// TIA Portal V20 export
FUNCTION "CallManualOperationLines_Unit1" : Void   // FC69, LAD
// stored: SetENOAutomatically false
   VAR_TEMP
      StatusEm : Array[0..7] of Struct
         Status : Array[0..45] of Word;
      END_STRUCT;
      errorIDEm : Array[0..7] of Struct
         errorID : Array[0..45] of Word;
      END_STRUCT;
      disableUnit1 : Bool;
      TempAxisCommands : "LBC_typeAxis64PosManualCommands";
      TempAxisMonitoring : "LBC_typeAxis64PosProcessValues";
      TempSoftCam : Array[0..8] of "LER_typeSoftCamParameter";
   END_VAR
   VAR CONSTANT
      MECHANIC_NAME_ENABLE : Bool;
   END_VAR
BEGIN

REGION Network 1: Unit 1 Enable Manual Operation
   // Condition to disable manual operation lines in Unit 1
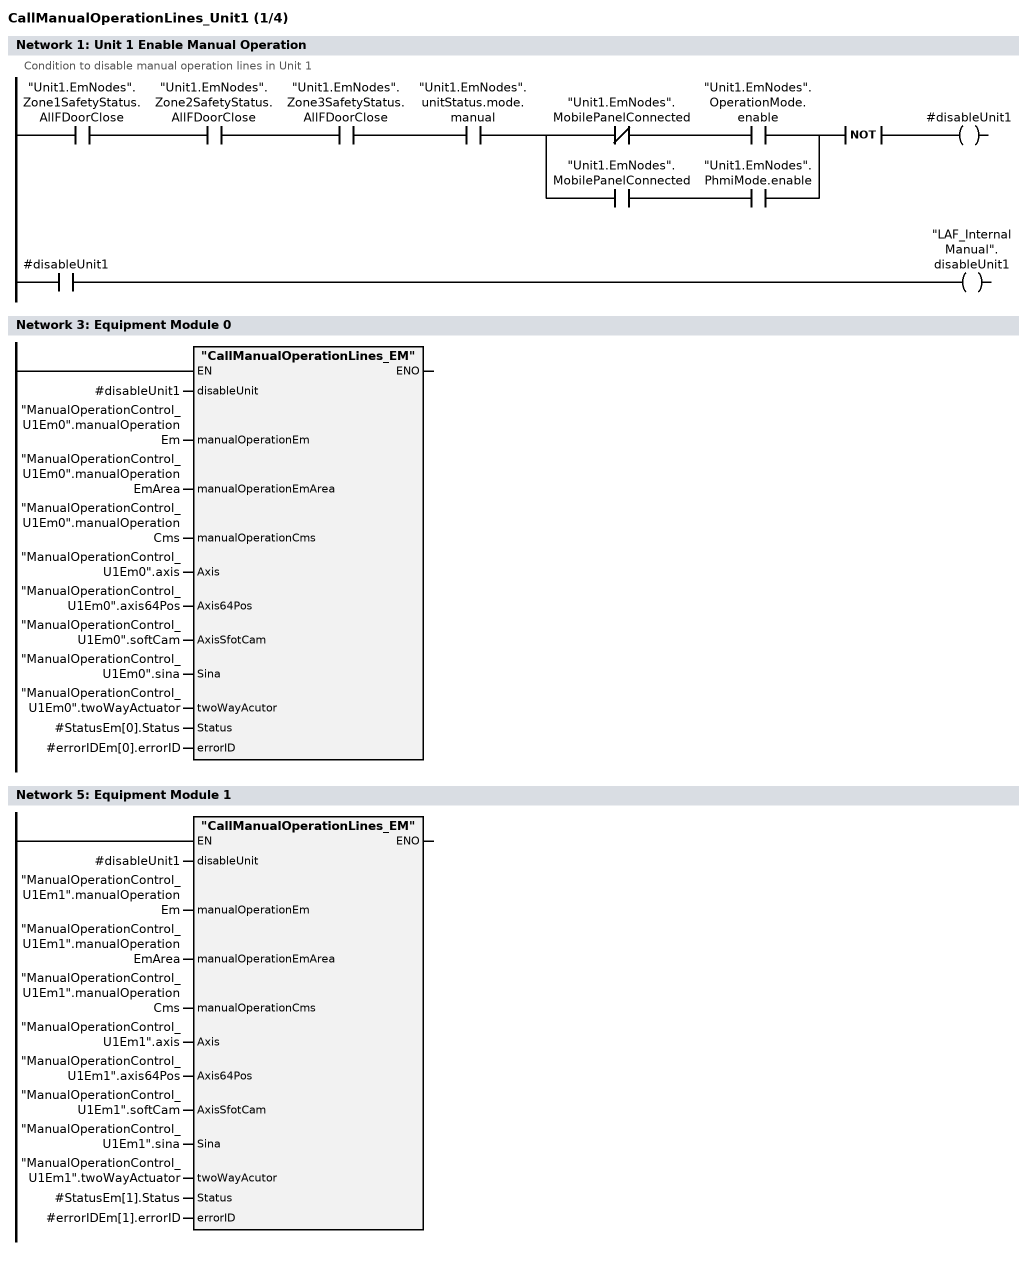
   RUNG wire#powerrail
      Contact( "Unit1.EmNodes".Zone1SafetyStatus.AllFDoorClose )
      Contact( "Unit1.EmNodes".Zone2SafetyStatus.AllFDoorClose )
      Contact( "Unit1.EmNodes".Zone3SafetyStatus.AllFDoorClose )
      Contact( "Unit1.EmNodes".unitStatus.mode.manual )
      wire#w1
      I_Contact( "Unit1.EmNodes".MobilePanelConnected )
      Contact( "Unit1.EmNodes".OperationMode.enable )
      wire#w2
      Not()
      Coil( #disableUnit1 )
   END_RUNG
   RUNG wire#w1
      Contact( "Unit1.EmNodes".MobilePanelConnected )
      Contact( "Unit1.EmNodes".PhmiMode.enable )
   END_RUNG wire#w2
   RUNG wire#powerrail
      Contact( #disableUnit1 )
      Coil( "LAF_InternalManual".disableUnit1 )
   END_RUNG
   // the same network as SCL:
   #disableUnit1 := NOT ("Unit1.EmNodes".Zone1SafetyStatus.AllFDoorClose AND "Unit1.EmNodes".Zone2SafetyStatus.AllFDoorClose AND "Unit1.EmNodes".Zone3SafetyStatus.AllFDoorClose AND "Unit1.EmNodes".unitStatus.mode.manual AND ((NOT "Unit1.EmNodes".MobilePanelConnected AND "Unit1.EmNodes".OperationMode.enable) OR ("Unit1.EmNodes".MobilePanelConnected AND "Unit1.EmNodes".PhmiMode.enable)));
   "LAF_InternalManual".disableUnit1 := #disableUnit1;
END_REGION

REGION Network 2 (SCL): Equipment Module 0 Cms Mapping
   REGION Input Mapping
       // Axis
       "ManualOperationControl_U1Em0".axis[1].monitoring := "Unit1.Em0.HmiInterface".cmUnWinderAxisB.monitoring;

       // TwoWayActuator
       "ManualOperationControl_U1Em0".twoWayActuator[1].monitoring := "Unit1.Em0.HmiInterface".cmAirShaftOnOff.monitoring;
       "ManualOperationControl_U1Em0".twoWayActuator[2].monitoring := "Unit1.Em0.HmiInterface".cmExpelFwdBwd.monitoring;
   END_REGION


   REGION Output Mapping
       // Axis
       "CallManualOperationLines_ServoCommands"(ManualOperationControl := "ManualOperationControl_U1Em0".axis[1].commands,
                                                HmiInterface => "Unit1.Em0.HmiInterface".cmUnWinderAxisB.commands);

       // TwoWayActuator
       "Unit1.Em0.HmiInterface".cmAirShaftOnOff.commands := "ManualOperationControl_U1Em0".twoWayActuator[1].commands;
       "Unit1.Em0.HmiInterface".cmExpelFwdBwd.commands := "ManualOperationControl_U1Em0".twoWayActuator[2].commands;
   END_REGION
END_REGION

REGION Network 3: Equipment Module 0
   RUNG wire#powerrail
      "CallManualOperationLines_EM"(disableUnit := #disableUnit1, manualOperationEm := "ManualOperationControl_U1Em0".manualOperationEm, manualOperationEmArea := "ManualOperationControl_U1Em0".manualOperationEmArea, manualOperationCms := "ManualOperationControl_U1Em0".manualOperationCms, Axis := "ManualOperationControl_U1Em0".axis, Axis64Pos := "ManualOperationControl_U1Em0".axis64Pos, AxisSfotCam := "ManualOperationControl_U1Em0".softCam, Sina := "ManualOperationControl_U1Em0".sina, twoWayAcutor := "ManualOperationControl_U1Em0".twoWayActuator, Status := #StatusEm[0].Status, errorID := #errorIDEm[0].errorID)
   END_RUNG
   // the same network as SCL:
   "CallManualOperationLines_EM"(disableUnit := #disableUnit1,
                           manualOperationEm := "ManualOperationControl_U1Em0".manualOperationEm,
                           manualOperationEmArea := "ManualOperationControl_U1Em0".manualOperationEmArea,
                           manualOperationCms := "ManualOperationControl_U1Em0".manualOperationCms,
                           Axis := "ManualOperationControl_U1Em0".axis,
                           Axis64Pos := "ManualOperationControl_U1Em0".axis64Pos,
                           AxisSfotCam := "ManualOperationControl_U1Em0".softCam,
                           Sina := "ManualOperationControl_U1Em0".sina,
                           twoWayAcutor := "ManualOperationControl_U1Em0".twoWayActuator,
                           Status := #StatusEm[0].Status,
                           errorID := #errorIDEm[0].errorID);
END_REGION

REGION Network 4 (SCL): Equipment Module 1 Cms Mapping
   REGION Input Mapping
       // Axis
       "ManualOperationControl_U1Em1".axis[1].monitoring := "Unit1.Em1.HmiInterface".cmUnWinderAxisB.monitoring;

       // TwoWayActuator
       "ManualOperationControl_U1Em1".twoWayActuator[1].monitoring := "Unit1.Em1.HmiInterface".cmAirShaftOnOff.monitoring;
       "ManualOperationControl_U1Em1".twoWayActuator[2].monitoring := "Unit1.Em1.HmiInterface".cmExpelFwdBwd.monitoring;
   END_REGION


   REGION Output Mapping
       // Axis
       "CallManualOperationLines_ServoCommands"(ManualOperationControl := "ManualOperationControl_U1Em1".axis[1].commands,
                                                HmiInterface => "Unit1.Em1.HmiInterface".cmUnWinderAxisB.commands);

       // TwoWayActuator
       "Unit1.Em1.HmiInterface".cmAirShaftOnOff.commands := "ManualOperationControl_U1Em1".twoWayActuator[1].commands;
       "Unit1.Em1.HmiInterface".cmExpelFwdBwd.commands := "ManualOperationControl_U1Em1".twoWayActuator[2].commands;
   END_REGION
END_REGION

REGION Network 5: Equipment Module 1
   RUNG wire#powerrail
      "CallManualOperationLines_EM"(disableUnit := #disableUnit1, manualOperationEm := "ManualOperationControl_U1Em1".manualOperationEm, manualOperationEmArea := "ManualOperationControl_U1Em1".manualOperationEmArea, manualOperationCms := "ManualOperationControl_U1Em1".manualOperationCms, Axis := "ManualOperationControl_U1Em1".axis, Axis64Pos := "ManualOperationControl_U1Em1".axis64Pos, AxisSfotCam := "ManualOperationControl_U1Em1".softCam, Sina := "ManualOperationControl_U1Em1".sina, twoWayAcutor := "ManualOperationControl_U1Em1".twoWayActuator, Status := #StatusEm[1].Status, errorID := #errorIDEm[1].errorID)
   END_RUNG
   // the same network as SCL:
   "CallManualOperationLines_EM"(disableUnit := #disableUnit1,
                           manualOperationEm := "ManualOperationControl_U1Em1".manualOperationEm,
                           manualOperationEmArea := "ManualOperationControl_U1Em1".manualOperationEmArea,
                           manualOperationCms := "ManualOperationControl_U1Em1".manualOperationCms,
                           Axis := "ManualOperationControl_U1Em1".axis,
                           Axis64Pos := "ManualOperationControl_U1Em1".axis64Pos,
                           AxisSfotCam := "ManualOperationControl_U1Em1".softCam,
                           Sina := "ManualOperationControl_U1Em1".sina,
                           twoWayAcutor := "ManualOperationControl_U1Em1".twoWayActuator,
                           Status := #StatusEm[1].Status,
                           errorID := #errorIDEm[1].errorID);
END_REGION

REGION Network 6 (SCL): Equipment Module 2 Cms Mapping
   REGION Input Mapping
       // TwoWayActuator
       "ManualOperationControl_U1Em2".twoWayActuator[1].monitoring := "Unit1.Em2.HmiInterface".cmElectrodeFixRightTopFwdBwd.monitoring;
       "ManualOperationControl_U1Em2".twoWayActuator[2].monitoring := "Unit1.Em2.HmiInterface".cmElectrodeFixRightBottomFwdBwd.monitoring;
       "ManualOperationControl_U1Em2".twoWayActuator[3].monitoring := "Unit1.Em2.HmiInterface".cmElectrodeFixLeftTopFwdBwd.monitoring;
       "ManualOperationControl_U1Em2".twoWayActuator[4].monitoring := "Unit1.Em2.HmiInterface".cmElectrodeFixLeftBottomFwdBwd.monitoring;
       "ManualOperationControl_U1Em2".twoWayActuator[5].monitoring := "Unit1.Em2.HmiInterface".cmElectrodeFixLeftTopUpDown.monitoring;
       "ManualOperationControl_U1Em2".twoWayActuator[6].monitoring := "Unit1.Em2.HmiInterface".cmElectrodeFixLeftBottomUpDown.monitoring;
       "ManualOperationControl_U1Em2".twoWayActuator[7].monitoring := "Unit1.Em2.HmiInterface".cmUwSemiSplicerVacuumRightTopOnOff.monitoring;
       "ManualOperationControl_U1Em2".twoWayActuator[8].monitoring := "Unit1.Em2.HmiInterface".cmUwSemiSplicerVacuumRightBottomOnOff.monitoring;
       "ManualOperationControl_U1Em2".twoWayActuator[9].monitoring := "Unit1.Em2.HmiInterface".cmUwSemiSplicerVacuumLeftTopOnOff.monitoring;
       "ManualOperationControl_U1Em2".twoWayActuator[10].monitoring := "Unit1.Em2.HmiInterface".cmUwSemiSplicerVacuumLeftBottomOnOff.monitoring;
       "ManualOperationControl_U1Em2".twoWayActuator[11].monitoring := "Unit1.Em2.HmiInterface".cmElectrodeCutterFwdBwd.monitoring;
       "ManualOperationControl_U1Em2".twoWayActuator[12].monitoring := "Unit1.Em2.HmiInterface".cmSplicingLeftModuleMoverFwdBwd.monitoring;
       "ManualOperationControl_U1Em2".twoWayActuator[13].monitoring := "Unit1.Em2.HmiInterface".cmSplicingRightModuleMoverFwdBwd.monitoring;
       "ManualOperationControl_U1Em2".twoWayActuator[14].monitoring := "Unit1.Em2.HmiInterface".cmElectrodeLeftHolderMoverFwdBwd.monitoring;
       "ManualOperationControl_U1Em2".twoWayActuator[15].monitoring := "Unit1.Em2.HmiInterface".cmElectrodeRightHolderMoverFwdBwd.monitoring;
       "ManualOperationControl_U1Em2".twoWayActuator[16].monitoring := "Unit1.Em2.HmiInterface".cmTapeLoadingTurnCwCcw.monitoring;
       "ManualOperationControl_U1Em2".twoWayActuator[17].monitoring := "Unit1.Em2.HmiInterface".cmTapeAttachUnitFwdBwd.monitoring;
       "ManualOperationControl_U1Em2".twoWayActuator[18].monitoring := "Unit1.Em2.HmiInterface".cmTapeVacuumOnOff.monitoring;
       "ManualOperationControl_U1Em2".twoWayActuator[19].monitoring := "Unit1.Em2.HmiInterface".cmStopperFwdBwd.monitoring;
       "ManualOperationControl_U1Em2".twoWayActuator[20].monitoring := "Unit1.Em2.HmiInterface".cmSupportUnitTransferFwdBwd.monitoring;
       "ManualOperationControl_U1Em2".twoWayActuator[21].monitoring := "Unit1.Em2.HmiInterface".cmSupportUnitShaftUpDown.monitoring;
       "ManualOperationControl_U1Em2".twoWayActuator[22].monitoring := "Unit1.Em2.HmiInterface".cmFrameCoverFwdBwd.monitoring;
   END_REGION


   REGION Output Mapping
       // TwoWayActuator
       "Unit1.Em2.HmiInterface".cmElectrodeFixRightTopFwdBwd.commands := "ManualOperationControl_U1Em2".twoWayActuator[1].commands;
       "Unit1.Em2.HmiInterface".cmElectrodeFixRightBottomFwdBwd.commands := "ManualOperationControl_U1Em2".twoWayActuator[2].commands;
       "Unit1.Em2.HmiInterface".cmElectrodeFixLeftTopFwdBwd.commands := "ManualOperationControl_U1Em2".twoWayActuator[3].commands;
       "Unit1.Em2.HmiInterface".cmElectrodeFixLeftBottomFwdBwd.commands := "ManualOperationControl_U1Em2".twoWayActuator[4].commands;
       "Unit1.Em2.HmiInterface".cmElectrodeFixLeftTopUpDown.commands := "ManualOperationControl_U1Em2".twoWayActuator[5].commands;
       "Unit1.Em2.HmiInterface".cmElectrodeFixLeftBottomUpDown.commands := "ManualOperationControl_U1Em2".twoWayActuator[6].commands;
       "Unit1.Em2.HmiInterface".cmUwSemiSplicerVacuumRightTopOnOff.commands := "ManualOperationControl_U1Em2".twoWayActuator[7].commands;
       "Unit1.Em2.HmiInterface".cmUwSemiSplicerVacuumRightBottomOnOff.commands := "ManualOperationControl_U1Em2".twoWayActuator[8].commands;
       "Unit1.Em2.HmiInterface".cmUwSemiSplicerVacuumLeftTopOnOff.commands := "ManualOperationControl_U1Em2".twoWayActuator[9].commands;
       "Unit1.Em2.HmiInterface".cmUwSemiSplicerVacuumLeftBottomOnOff.commands := "ManualOperationControl_U1Em2".twoWayActuator[10].commands;
       "Unit1.Em2.HmiInterface".cmElectrodeCutterFwdBwd.commands := "ManualOperationControl_U1Em2".twoWayActuator[11].commands;
       "Unit1.Em2.HmiInterface".cmSplicingLeftModuleMoverFwdBwd.commands := "ManualOperationControl_U1Em2".twoWayActuator[12].commands;
       "Unit1.Em2.HmiInterface".cmSplicingRightModuleMoverFwdBwd.commands := "ManualOperationControl_U1Em2".twoWayActuator[13].commands;
       "Unit1.Em2.HmiInterface".cmElectrodeLeftHolderMoverFwdBwd.commands := "ManualOperationControl_U1Em2".twoWayActuator[14].commands;
       "Unit1.Em2.HmiInterface".cmElectrodeRightHolderMoverFwdBwd.commands := "ManualOperationControl_U1Em2".twoWayActuator[15].commands;
       "Unit1.Em2.HmiInterface".cmTapeLoadingTurnCwCcw.commands := "ManualOperationControl_U1Em2".twoWayActuator[16].commands;
       "Unit1.Em2.HmiInterface".cmTapeAttachUnitFwdBwd.commands := "ManualOperationControl_U1Em2".twoWayActuator[17].commands;
       "Unit1.Em2.HmiInterface".cmTapeVacuumOnOff.commands := "ManualOperationControl_U1Em2".twoWayActuator[18].commands;
       "Unit1.Em2.HmiInterface".cmStopperFwdBwd.commands := "ManualOperationControl_U1Em2".twoWayActuator[19].commands;
       "Unit1.Em2.HmiInterface".cmSupportUnitTransferFwdBwd.commands := "ManualOperationControl_U1Em2".twoWayActuator[20].commands;
       "Unit1.Em2.HmiInterface".cmSupportUnitShaftUpDown.commands := "ManualOperationControl_U1Em2".twoWayActuator[21].commands;
       "Unit1.Em2.HmiInterface".cmFrameCoverFwdBwd.commands := "ManualOperationControl_U1Em2".twoWayActuator[22].commands;
   END_REGION
END_REGION

REGION Network 7: Equipment Module 2
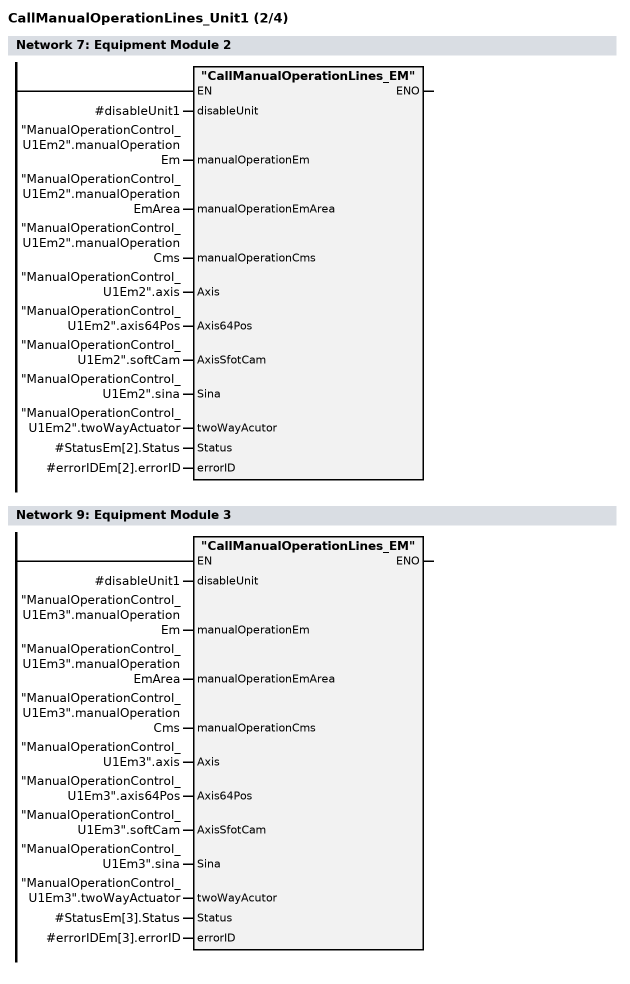
   RUNG wire#powerrail
      "CallManualOperationLines_EM"(disableUnit := #disableUnit1, manualOperationEm := "ManualOperationControl_U1Em2".manualOperationEm, manualOperationEmArea := "ManualOperationControl_U1Em2".manualOperationEmArea, manualOperationCms := "ManualOperationControl_U1Em2".manualOperationCms, Axis := "ManualOperationControl_U1Em2".axis, Axis64Pos := "ManualOperationControl_U1Em2".axis64Pos, AxisSfotCam := "ManualOperationControl_U1Em2".softCam, Sina := "ManualOperationControl_U1Em2".sina, twoWayAcutor := "ManualOperationControl_U1Em2".twoWayActuator, Status := #StatusEm[2].Status, errorID := #errorIDEm[2].errorID)
   END_RUNG
   // the same network as SCL:
   "CallManualOperationLines_EM"(disableUnit := #disableUnit1,
                           manualOperationEm := "ManualOperationControl_U1Em2".manualOperationEm,
                           manualOperationEmArea := "ManualOperationControl_U1Em2".manualOperationEmArea,
                           manualOperationCms := "ManualOperationControl_U1Em2".manualOperationCms,
                           Axis := "ManualOperationControl_U1Em2".axis,
                           Axis64Pos := "ManualOperationControl_U1Em2".axis64Pos,
                           AxisSfotCam := "ManualOperationControl_U1Em2".softCam,
                           Sina := "ManualOperationControl_U1Em2".sina,
                           twoWayAcutor := "ManualOperationControl_U1Em2".twoWayActuator,
                           Status := #StatusEm[2].Status,
                           errorID := #errorIDEm[2].errorID);
END_REGION

REGION Network 8 (SCL): Equipment Module 3 Cms Mapping
   REGION Input Mapping
       // TwoWayActuator
       "ManualOperationControl_U1Em3".twoWayActuator[1].monitoring := "Unit1.Em3.HmiInterface".cmDancerRegulatorOnOff.monitoring;
   END_REGION


   REGION Output Mapping
       // TwoWayActuator
       "Unit1.Em3.HmiInterface".cmDancerRegulatorOnOff.commands := "ManualOperationControl_U1Em3".twoWayActuator[1].commands;
   END_REGION
END_REGION

REGION Network 9: Equipment Module 3
   RUNG wire#powerrail
      "CallManualOperationLines_EM"(disableUnit := #disableUnit1, manualOperationEm := "ManualOperationControl_U1Em3".manualOperationEm, manualOperationEmArea := "ManualOperationControl_U1Em3".manualOperationEmArea, manualOperationCms := "ManualOperationControl_U1Em3".manualOperationCms, Axis := "ManualOperationControl_U1Em3".axis, Axis64Pos := "ManualOperationControl_U1Em3".axis64Pos, AxisSfotCam := "ManualOperationControl_U1Em3".softCam, Sina := "ManualOperationControl_U1Em3".sina, twoWayAcutor := "ManualOperationControl_U1Em3".twoWayActuator, Status := #StatusEm[3].Status, errorID := #errorIDEm[3].errorID)
   END_RUNG
   // the same network as SCL:
   "CallManualOperationLines_EM"(disableUnit := #disableUnit1,
                           manualOperationEm := "ManualOperationControl_U1Em3".manualOperationEm,
                           manualOperationEmArea := "ManualOperationControl_U1Em3".manualOperationEmArea,
                           manualOperationCms := "ManualOperationControl_U1Em3".manualOperationCms,
                           Axis := "ManualOperationControl_U1Em3".axis,
                           Axis64Pos := "ManualOperationControl_U1Em3".axis64Pos,
                           AxisSfotCam := "ManualOperationControl_U1Em3".softCam,
                           Sina := "ManualOperationControl_U1Em3".sina,
                           twoWayAcutor := "ManualOperationControl_U1Em3".twoWayActuator,
                           Status := #StatusEm[3].Status,
                           errorID := #errorIDEm[3].errorID);
END_REGION

REGION Network 10 (SCL): Equipment Module 4 Cms Mapping
   REGION Input Mapping
       // Axis
       "ManualOperationControl_U1Em4".axis[1].monitoring := "Unit1.Em4.HmiInterface".cmCompensatorAxisZ.monitoring;
       "ManualOperationControl_U1Em4".axis[2].monitoring := "Unit1.Em4.HmiInterface".cmFeedingRollAxisB.monitoring;
       "ManualOperationControl_U1Em4".axis[3].monitoring := "Unit1.Em4.HmiInterface".cmElectrodeCutterAxisZ.monitoring;
       "ManualOperationControl_U1Em4".axis64Pos[1].monitoring := "Unit1.Em4.HmiInterface".cmPositionMovingAxisX.monitoring;

       // SoftCam
       "ManualOperationControl_U1Em4".softCam[1] := "Unit1.Em4.HmiInterface".cm.softcam.positionMoving;

       // TwoWayActuator
       "ManualOperationControl_U1Em4".twoWayActuator[1].monitoring := "Unit1.Em4.HmiInterface".cmFeederCylinderUpDown.monitoring;
   END_REGION


   REGION Output Mapping
       // Axis
       "CallManualOperationLines_ServoCommands"(ManualOperationControl := "ManualOperationControl_U1Em4".axis[1].commands,
                                                HmiInterface => "Unit1.Em4.HmiInterface".cmCompensatorAxisZ.commands);
       "CallManualOperationLines_ServoCommands"(ManualOperationControl := "ManualOperationControl_U1Em4".axis[2].commands,
                                                HmiInterface => "Unit1.Em4.HmiInterface".cmFeedingRollAxisB.commands);
       "CallManualOperationLines_ServoCommands"(ManualOperationControl := "ManualOperationControl_U1Em4".axis[3].commands,
                                                HmiInterface => "Unit1.Em4.HmiInterface".cmElectrodeCutterAxisZ.commands);
       "CallManualOperationLines_ServoPos64Commands"(ManualOperationControl := "ManualOperationControl_U1Em4".axis64Pos[1].commands,
                                                     HmiInterface => "Unit1.Em4.HmiInterface".cmPositionMovingAxisX.commands);

       // TwoWayActuator
       "Unit1.Em4.HmiInterface".cmFeederCylinderUpDown.commands := "ManualOperationControl_U1Em4".twoWayActuator[1].commands;
   END_REGION
END_REGION

REGION Network 11: Equipment Module 4
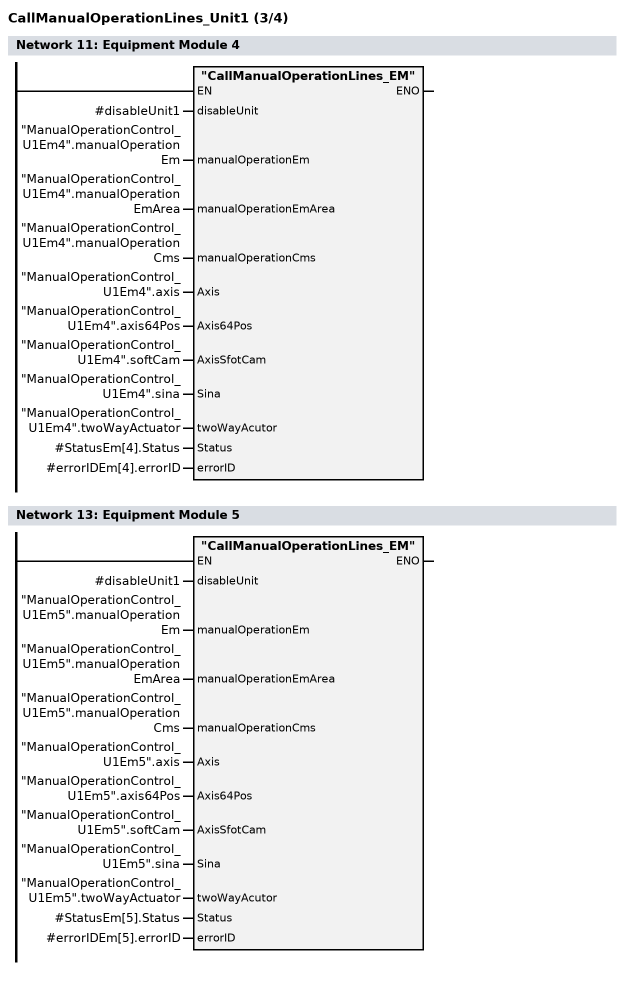
   RUNG wire#powerrail
      "CallManualOperationLines_EM"(disableUnit := #disableUnit1, manualOperationEm := "ManualOperationControl_U1Em4".manualOperationEm, manualOperationEmArea := "ManualOperationControl_U1Em4".manualOperationEmArea, manualOperationCms := "ManualOperationControl_U1Em4".manualOperationCms, Axis := "ManualOperationControl_U1Em4".axis, Axis64Pos := "ManualOperationControl_U1Em4".axis64Pos, AxisSfotCam := "ManualOperationControl_U1Em4".softCam, Sina := "ManualOperationControl_U1Em4".sina, twoWayAcutor := "ManualOperationControl_U1Em4".twoWayActuator, Status := #StatusEm[4].Status, errorID := #errorIDEm[4].errorID)
   END_RUNG
   // the same network as SCL:
   "CallManualOperationLines_EM"(disableUnit := #disableUnit1,
                           manualOperationEm := "ManualOperationControl_U1Em4".manualOperationEm,
                           manualOperationEmArea := "ManualOperationControl_U1Em4".manualOperationEmArea,
                           manualOperationCms := "ManualOperationControl_U1Em4".manualOperationCms,
                           Axis := "ManualOperationControl_U1Em4".axis,
                           Axis64Pos := "ManualOperationControl_U1Em4".axis64Pos,
                           AxisSfotCam := "ManualOperationControl_U1Em4".softCam,
                           Sina := "ManualOperationControl_U1Em4".sina,
                           twoWayAcutor := "ManualOperationControl_U1Em4".twoWayActuator,
                           Status := #StatusEm[4].Status,
                           errorID := #errorIDEm[4].errorID);
END_REGION

REGION Network 12 (SCL): Equipment Module 5 Cms Mapping
   REGION Input Mapping
       // Axis
       "ManualOperationControl_U1Em5".axis64Pos[1].monitoring := "Unit1.Em5.HmiInterface".cmNgAndManualInputAxisY.monitoring;
       "ManualOperationControl_U1Em5".axis64Pos[2].monitoring := "Unit1.Em5.HmiInterface".cmMagazineAxisZ.monitoring;

       // SoftCam
       "ManualOperationControl_U1Em5".softCam[1] := "Unit1.Em5.HmiInterface".cm.softcam.ngAndManualInput;
       "ManualOperationControl_U1Em5".softCam[2] := "Unit1.Em5.HmiInterface".cm.softcam.magazine;

       // TwoWayActuator
       "ManualOperationControl_U1Em5".twoWayActuator[1].monitoring := "Unit1.Em5.HmiInterface".cmNgAndManualInputCylinderUpDown.monitoring;
       "ManualOperationControl_U1Em5".twoWayActuator[2].monitoring := "Unit1.Em5.HmiInterface".cmNgAndManualInputVacuum1OnOff.monitoring;
       "ManualOperationControl_U1Em5".twoWayActuator[3].monitoring := "Unit1.Em5.HmiInterface".cmNgAndManualInputVacuum2OnOff.monitoring;
       "ManualOperationControl_U1Em5".twoWayActuator[4].monitoring := "Unit1.Em5.HmiInterface".cmNgAndManualInputVibrator1OnOff.monitoring;
       "ManualOperationControl_U1Em5".twoWayActuator[5].monitoring := "Unit1.Em5.HmiInterface".cmNgAndManualInputVibrator2OnOff.monitoring;
       "ManualOperationControl_U1Em5".twoWayActuator[6].monitoring := "Unit1.Em5.HmiInterface".cmMagazineLockCylinderUpDown.monitoring;
   END_REGION


   REGION Output Mapping
       // Axis
       "CallManualOperationLines_ServoPos64Commands"(ManualOperationControl := "ManualOperationControl_U1Em5".axis64Pos[1].commands,
                                                     HmiInterface => "Unit1.Em5.HmiInterface".cmNgAndManualInputAxisY.commands);
       "CallManualOperationLines_ServoPos64Commands"(ManualOperationControl := "ManualOperationControl_U1Em5".axis64Pos[2].commands,
                                                     HmiInterface => "Unit1.Em5.HmiInterface".cmMagazineAxisZ.commands);

       // TwoWayActuator
       "Unit1.Em5.HmiInterface".cmNgAndManualInputCylinderUpDown.commands := "ManualOperationControl_U1Em5".twoWayActuator[1].commands;
       "Unit1.Em5.HmiInterface".cmNgAndManualInputVacuum1OnOff.commands := "ManualOperationControl_U1Em5".twoWayActuator[2].commands;
       "Unit1.Em5.HmiInterface".cmNgAndManualInputVacuum2OnOff.commands := "ManualOperationControl_U1Em5".twoWayActuator[3].commands;
       "Unit1.Em5.HmiInterface".cmNgAndManualInputVibrator1OnOff.commands := "ManualOperationControl_U1Em5".twoWayActuator[4].commands;
       "Unit1.Em5.HmiInterface".cmNgAndManualInputVibrator2OnOff.commands := "ManualOperationControl_U1Em5".twoWayActuator[5].commands;
       "Unit1.Em5.HmiInterface".cmMagazineLockCylinderUpDown.commands := "ManualOperationControl_U1Em5".twoWayActuator[6].commands;
   END_REGION
END_REGION

REGION Network 13: Equipment Module 5
   RUNG wire#powerrail
      "CallManualOperationLines_EM"(disableUnit := #disableUnit1, manualOperationEm := "ManualOperationControl_U1Em5".manualOperationEm, manualOperationEmArea := "ManualOperationControl_U1Em5".manualOperationEmArea, manualOperationCms := "ManualOperationControl_U1Em5".manualOperationCms, Axis := "ManualOperationControl_U1Em5".axis, Axis64Pos := "ManualOperationControl_U1Em5".axis64Pos, AxisSfotCam := "ManualOperationControl_U1Em5".softCam, Sina := "ManualOperationControl_U1Em5".sina, twoWayAcutor := "ManualOperationControl_U1Em5".twoWayActuator, Status := #StatusEm[5].Status, errorID := #errorIDEm[5].errorID)
   END_RUNG
   // the same network as SCL:
   "CallManualOperationLines_EM"(disableUnit := #disableUnit1,
                           manualOperationEm := "ManualOperationControl_U1Em5".manualOperationEm,
                           manualOperationEmArea := "ManualOperationControl_U1Em5".manualOperationEmArea,
                           manualOperationCms := "ManualOperationControl_U1Em5".manualOperationCms,
                           Axis := "ManualOperationControl_U1Em5".axis,
                           Axis64Pos := "ManualOperationControl_U1Em5".axis64Pos,
                           AxisSfotCam := "ManualOperationControl_U1Em5".softCam,
                           Sina := "ManualOperationControl_U1Em5".sina,
                           twoWayAcutor := "ManualOperationControl_U1Em5".twoWayActuator,
                           Status := #StatusEm[5].Status,
                           errorID := #errorIDEm[5].errorID);
END_REGION

REGION Network 14 (SCL): Equipment Module 6 Cms Mapping
   REGION Input Mapping
       // Axis
       "ManualOperationControl_U1Em6".axis64Pos[1].monitoring := "Unit1.Em6.HmiInterface".cmVisionUnitAxisZ.monitoring;

       // SoftCam
       "ManualOperationControl_U1Em6".softCam[1] := "Unit1.Em6.HmiInterface".cm.softcam.visionUnit;

       // TwoWayActuator
       "ManualOperationControl_U1Em6".twoWayActuator[1].monitoring := "Unit1.Em6.HmiInterface".cmVisionPusherSupportUpDown.monitoring;
   END_REGION


   REGION Output Mapping
       // Axis
       "CallManualOperationLines_ServoPos64Commands"(ManualOperationControl := "ManualOperationControl_U1Em6".axis64Pos[1].commands,
                                                     HmiInterface => "Unit1.Em6.HmiInterface".cmVisionUnitAxisZ.commands);

       // TwoWayActuator
       "Unit1.Em6.HmiInterface".cmVisionPusherSupportUpDown.commands := "ManualOperationControl_U1Em6".twoWayActuator[1].commands;
   END_REGION
END_REGION

REGION Network 15: Equipment Module 6
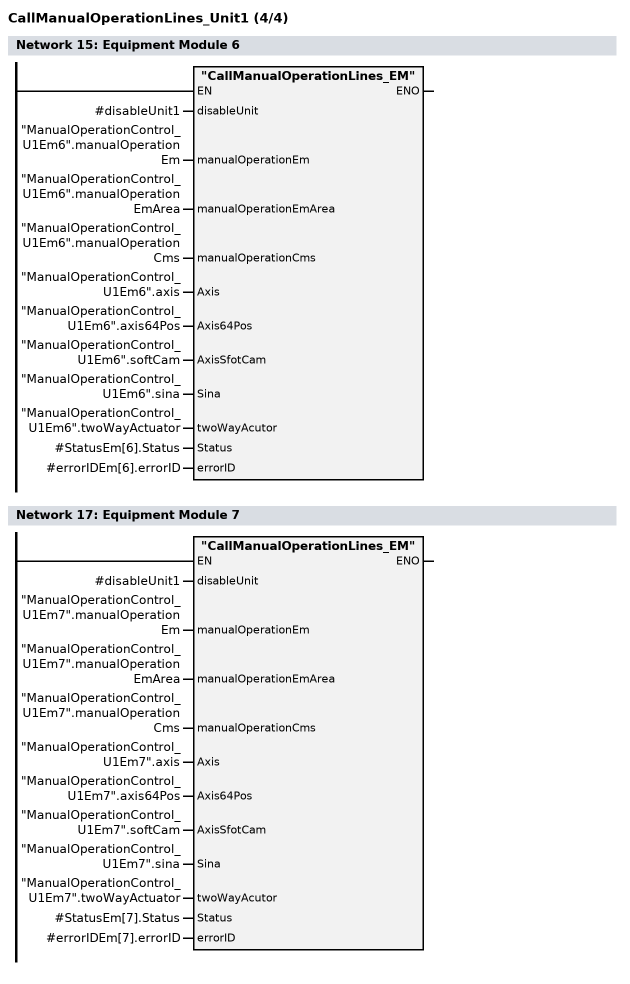
   RUNG wire#powerrail
      "CallManualOperationLines_EM"(disableUnit := #disableUnit1, manualOperationEm := "ManualOperationControl_U1Em6".manualOperationEm, manualOperationEmArea := "ManualOperationControl_U1Em6".manualOperationEmArea, manualOperationCms := "ManualOperationControl_U1Em6".manualOperationCms, Axis := "ManualOperationControl_U1Em6".axis, Axis64Pos := "ManualOperationControl_U1Em6".axis64Pos, AxisSfotCam := "ManualOperationControl_U1Em6".softCam, Sina := "ManualOperationControl_U1Em6".sina, twoWayAcutor := "ManualOperationControl_U1Em6".twoWayActuator, Status := #StatusEm[6].Status, errorID := #errorIDEm[6].errorID)
   END_RUNG
   // the same network as SCL:
   "CallManualOperationLines_EM"(disableUnit := #disableUnit1,
                           manualOperationEm := "ManualOperationControl_U1Em6".manualOperationEm,
                           manualOperationEmArea := "ManualOperationControl_U1Em6".manualOperationEmArea,
                           manualOperationCms := "ManualOperationControl_U1Em6".manualOperationCms,
                           Axis := "ManualOperationControl_U1Em6".axis,
                           Axis64Pos := "ManualOperationControl_U1Em6".axis64Pos,
                           AxisSfotCam := "ManualOperationControl_U1Em6".softCam,
                           Sina := "ManualOperationControl_U1Em6".sina,
                           twoWayAcutor := "ManualOperationControl_U1Em6".twoWayActuator,
                           Status := #StatusEm[6].Status,
                           errorID := #errorIDEm[6].errorID);
END_REGION

REGION Network 16 (SCL): Equipment Module 7 Cms Mapping
   REGION Input Mapping
       // Axis
       "ManualOperationControl_U1Em7".axis[1].monitoring := "Unit1.Em7.HmiInterface".cmNgKickerAxisZ.monitoring;
       "ManualOperationControl_U1Em7".axis[2].monitoring := "Unit1.Em7.HmiInterface".cmPassKickerAxisZ.monitoring;
       "ManualOperationControl_U1Em7".axis[3].monitoring := "Unit1.Em7.HmiInterface".cmCutConveyorAxisB.monitoring;
       "ManualOperationControl_U1Em7".axis[4].monitoring := "Unit1.Em7.HmiInterface".cmNgConveyorAxisB.monitoring;
       "ManualOperationControl_U1Em7".axis[5].monitoring := "Unit1.Em7.HmiInterface".cmStack1ConveyorAxisB.monitoring;
       "ManualOperationControl_U1Em7".axis[6].monitoring := "Unit1.Em7.HmiInterface".cmStack2ConveyorAxisB.monitoring;

       // Sina Speed
       "ManualOperationControl_U1Em7".sina[1].monitoring := "Unit1.Em7.HmiInterface".cmCutConveyorRingBlow.monitoring;
       "ManualOperationControl_U1Em7".sina[2].monitoring := "Unit1.Em7.HmiInterface".cmNgConveyorRingBlow.monitoring;
       "ManualOperationControl_U1Em7".sina[3].monitoring := "Unit1.Em7.HmiInterface".cmStack2ConveyorRingBlow.monitoring;

       // TwoWayActuator
       "ManualOperationControl_U1Em7".twoWayActuator[1].monitoring := "Unit1.Em7.HmiInterface".cmNgBoxLockCylinderUpDown.monitoring;
   END_REGION


   REGION Output Mapping
       // Axis
       "CallManualOperationLines_ServoCommands"(ManualOperationControl := "ManualOperationControl_U1Em7".axis[1].commands,
                                                HmiInterface => "Unit1.Em7.HmiInterface".cmNgKickerAxisZ.commands);
       "CallManualOperationLines_ServoCommands"(ManualOperationControl := "ManualOperationControl_U1Em7".axis[2].commands,
                                                HmiInterface => "Unit1.Em7.HmiInterface".cmPassKickerAxisZ.commands);
       "CallManualOperationLines_ServoCommands"(ManualOperationControl := "ManualOperationControl_U1Em7".axis[3].commands,
                                                HmiInterface => "Unit1.Em7.HmiInterface".cmCutConveyorAxisB.commands);
       "CallManualOperationLines_ServoCommands"(ManualOperationControl := "ManualOperationControl_U1Em7".axis[4].commands,
                                                HmiInterface => "Unit1.Em7.HmiInterface".cmNgConveyorAxisB.commands);
       "CallManualOperationLines_ServoCommands"(ManualOperationControl := "ManualOperationControl_U1Em7".axis[5].commands,
                                                HmiInterface => "Unit1.Em7.HmiInterface".cmStack1ConveyorAxisB.commands);
       "CallManualOperationLines_ServoCommands"(ManualOperationControl := "ManualOperationControl_U1Em7".axis[6].commands,
                                                HmiInterface => "Unit1.Em7.HmiInterface".cmStack2ConveyorAxisB.commands);

       // Sina Speed
       "Unit1.Em7.HmiInterface".cmCutConveyorRingBlow.commands.moveVelocity := "ManualOperationControl_U1Em7".sina[1].commands.moveVelocity;
       "Unit1.Em7.HmiInterface".cmCutConveyorRingBlow.commands.stop := "ManualOperationControl_U1Em7".sina[1].commands.stop;
       "Unit1.Em7.HmiInterface".cmNgConveyorRingBlow.commands.moveVelocity := "ManualOperationControl_U1Em7".sina[2].commands.moveVelocity;
       "Unit1.Em7.HmiInterface".cmNgConveyorRingBlow.commands.stop := "ManualOperationControl_U1Em7".sina[2].commands.stop;
       "Unit1.Em7.HmiInterface".cmStack2ConveyorRingBlow.commands.moveVelocity := "ManualOperationControl_U1Em7".sina[3].commands.moveVelocity;
       "Unit1.Em7.HmiInterface".cmStack2ConveyorRingBlow.commands.stop := "ManualOperationControl_U1Em7".sina[3].commands.stop;

       // TwoWayActuator
       "Unit1.Em7.HmiInterface".cmNgBoxLockCylinderUpDown.commands := "ManualOperationControl_U1Em7".twoWayActuator[1].commands;
   END_REGION
END_REGION

REGION Network 17: Equipment Module 7
   RUNG wire#powerrail
      "CallManualOperationLines_EM"(disableUnit := #disableUnit1, manualOperationEm := "ManualOperationControl_U1Em7".manualOperationEm, manualOperationEmArea := "ManualOperationControl_U1Em7".manualOperationEmArea, manualOperationCms := "ManualOperationControl_U1Em7".manualOperationCms, Axis := "ManualOperationControl_U1Em7".axis, Axis64Pos := "ManualOperationControl_U1Em7".axis64Pos, AxisSfotCam := "ManualOperationControl_U1Em7".softCam, Sina := "ManualOperationControl_U1Em7".sina, twoWayAcutor := "ManualOperationControl_U1Em7".twoWayActuator, Status := #StatusEm[7].Status, errorID := #errorIDEm[7].errorID)
   END_RUNG
   // the same network as SCL:
   "CallManualOperationLines_EM"(disableUnit := #disableUnit1,
                           manualOperationEm := "ManualOperationControl_U1Em7".manualOperationEm,
                           manualOperationEmArea := "ManualOperationControl_U1Em7".manualOperationEmArea,
                           manualOperationCms := "ManualOperationControl_U1Em7".manualOperationCms,
                           Axis := "ManualOperationControl_U1Em7".axis,
                           Axis64Pos := "ManualOperationControl_U1Em7".axis64Pos,
                           AxisSfotCam := "ManualOperationControl_U1Em7".softCam,
                           Sina := "ManualOperationControl_U1Em7".sina,
                           twoWayAcutor := "ManualOperationControl_U1Em7".twoWayActuator,
                           Status := #StatusEm[7].Status,
                           errorID := #errorIDEm[7].errorID);
END_REGION
END_FUNCTION
